Staubli VAL3: SockRec.pgx

public program SockRec(string& StrDatRec[] (dimensions=1), bool& stat[] (dimensions=1))
  local bool FdataR
  local num CharaS
  local num DataR
  local num SckStat
  local string Step1
  local string Strdata
  local string Strrec
  local string Scrdata1
begin
  //This program is being used to recieve the TCP data
  //Parameter description: StrDatRec--> data to be recieved in string type
  //                       stat----> bool value to tell the end of data recieving
  //Program can call this subroutine to recieve the data from tcp socket
  //In control panel , io:socket need be pre-defined
  // port 1000 , timeout :0 delimitier :1 TCP client name : socket
  sioLink(sock,socket)
  while true
    DataR=DataR+1
    CharaS=sioGet(sock,SckStat)
    Strrec=chr(SckStat)
    if Strrec=="("
      FdataR=true
    endIf
    if Strrec==")"
      FdataR=false
    endIf
    if FdataR==true
      Strdata=Strdata+Strrec
    else
      Scrdata1=Strdata
      if Scrdata1!=""
        StrDatRec=Scrdata1+")"
        stat=true
      else
        StrDatRec=""
      endIf
      Strdata=""
    endIf
    delay(0)
  endWhile
end
